# EPICS autosave request: QHYApp/Db/QHYDriver_settings.req
file "ADBase_settings.req", P=$(P), R=$(R)
$(P)$(R)Offset
$(P)$(R)ReadoutMode
$(P)$(R)ReadMode
